PROGRAM P_ProfilePositionModeTest
VAR
	fbMoveInProfilePosition			: Motion;
	fbGetCurrentPosition			: FB_EcCoeSdoRead;
	fbGetStatusword					: FB_EcCoeSdoRead;
	fbGetPositionWindow				: FB_EcCoeSdoRead;
	fbGetPositionDemandValue		: FB_EcCoeSdoRead;
	tWaitForCurrentPosition			: TON;
	tWaitForPositionDemandValue		: TON;
	tGetStatusword					: TON;
	bGetCurrentPosition				: BOOL;
	bMove							: BOOL; 
	bExecuteTimer					: BOOL;
	bGetStatusword					: BOOL;
	bGetParameters					: BOOL;
	bSetPositioningOptionCode		: BOOL;
	bGetPositionDemandValue			: BOOL;
	bBasicOperationAbsStarted		: BOOL;
	bBasicOperationAbsFinished		: BOOL := FALSE;
	bPositioningOptionCodeSet		: BOOL;
	bTargetReached					: BOOL;
	bTestAbsolutePositioning		: BOOL;
	nTargetPosition					: DINT;
	nCurrentPosition				: DINT;
	nTargetPositionBuf				: DINT;
	nPositionDemandValue			: DINT;
	nStatusword						: UINT;
	nPositionWindow					: UDINT;
	
	
	bTest							: BOOL;
	bAusprobieren					: BOOL;
END_VAR

VAR
	bBasicOperationAbs				: BOOL;
	bBasicOperationRel				: BOOL;
	bPositioningOptionCode			: BOOL;
END_VAR

//For Test Set of Setpoints
VAR
	bSetOfSetpointFinished 			: BOOL;
	nCurrentPositionBuf				: DINT;
	bSetPointSet					: BOOL;  //For both
	bSetOfSetpoints					: BOOL;
	bStartBasicOperationAbs			: BOOL;
	bTestSetOfSetpoints				: BOOL;
	bSetOfSetpointsFinished			: BOOL;
END_VAR

//Fo Test Change Immediately
VAR
	bTestChangeImmediately			: BOOL;
	bChangeImmediatelyFinished		: BOOL;
	bChangeImmediately				: BOOL;
END_VAR

//For test of relative Positioninig
VAR
	tSetPositioningOptionCode		: TON;
	fbSetPositioningOptionCode		: FB_EcCoeSdoWrite;
	bTestRelativePositioning		: BOOL;
	bRelativePositioningFinished	: BOOL;
	nPositioningOptionCode			: DINT;
	nCounter						: DINT;
END_VAR

tWaitForCurrentPosition(IN := bGetCurrentPosition,
							PT := T#10MS);
tGetStatusword(IN := bGetStatusword,
					PT := T#500MS);	
tSetPositioningOptionCode(IN := bSetPositioningOptionCode,
							PT := T#125MS);		
tWaitForPositionDemandValue(IN := bGetPositionDemandValue,
							PT := T#125MS);
IF tWaitForCurrentPosition.Q THEN
	bGetCurrentPosition := FALSE;
ELSE
	bGetCurrentPosition := TRUE;		
END_IF
fbMoveInProfilePosition(sNetID := GVL.sNetId,
						nSlaveAddr := GVL.nSlaveAddr,
						nTargetPosition := nTargetPosition,
						bMove := bMove);
fbGetStatusword(sNetId := GVL.sNetId,
				nSlaveAddr := GVL.nSlaveAddr,
				nIndex := 16#6041,
				nSubindex := 0,
				pDstBuf := ADR(nStatusWord),
				cbBufLen := SIZEOF(nStatusWord),
				bExecute := bGetStatusword);
fbGetCurrentPosition(sNetId := GVL.sNetId,
						nSlaveAddr := GVL.nSlaveAddr,
						nIndex := 16#6064,
						nSubIndex := 0,
						pDstBuf := ADR(nCurrentPosition),
						cbBufLen := SIZEOF(nCurrentPosition),
						bExecute := bGetCurrentPosition);
fbGetPositionWindow(sNetId := GVL.sNetId,
					nSlaveAddr := GVL.nSlaveAddr,
					nIndex := 16#6067,
					nSubIndex := 0,
					pDstBuf := ADR(nPositionWindow),
					cbBufLen := SIZEOF(nPositionWindow),
					bExecute := bGetParameters);
fbGetPositionDemandValue(sNetId := GVL.sNetId,
							nSlaveAddr := GVL.nSlaveAddr,
							nIndex := 16#60FC,
							nSubIndex := 0,
							pDstBuf := ADR(nPositionDemandValue),
							cbBufLen := SIZEOF(nPositionDemandValue),
							bExecute := bGetPositionDemandValue);
fbSetPositioningOptionCode(sNetId := GVL.sNetId,
							nSlaveAddr := GVL.nSlaveAddr,
							nIndex := 16#60F2,
							nSubindex := 0,
							pSrcBuf := ADR(nPositioningOptionCode),
							cbBufLen := SIZEOF(nPositioningOptionCode),
							bExecute := bSetPositioningOptionCode);
bGetParameters := TRUE;

IF bStartBasicOperationAbs THEN					
	//Basic Operation
	//Set-point is applied to the device
	//Move to absolute position is tested
	//Wait until Target reach Bit is set
	//Control if position is within error window
	
	//Target shall be an absolute value
	MAIN.Controlword.6 := 0;

	//Operation has not yet started and we are sure that initial position is obtained
	IF NOT bBasicOperationAbsStarted THEN
		nTargetPosition := nCurrentPosition + 5000000;
		//Start absolute positioning
		bMove := TRUE;	
		bBasicOperationAbsStarted := TRUE;
	END_IF
					
	//Target reached?
	bGetStatusword := TRUE;
	IF tGetStatusword.Q THEN
		IF NOT nStatusword.10 THEN
			bGetStatusword := FALSE;
		ELSIF ((nCurrentPosition >= nTargetPosition - nPositionWindow)
				AND (nCurrentPosition <= nTargetPosition + nPositionWindow)) 
				AND fbMoveInProfilePosition.bStartPositioning THEN
			//absolute Positionining
			bBasicOperationAbs := TRUE;
			bBasicOperationAbsFinished := TRUE;
			bStartBasicOperationAbs := FALSE;
		ELSIF fbMoveInProfilePosition.bStartPositioning THEN
			bBasicOperationAbs := FALSE;
			bBasicOperationAbsFinished := TRUE;
			bStartBasicOperationAbs := FALSE;
		END_IF
		bGetStatusword := FALSE;
	END_IF
END_IF

//Test SetOfSetpoints
IF bTestSetOfSetpoints AND bBasicOperationAbsFinished AND NOT bSetOfSetpointsFinished THEN
	IF NOT bSetPointSet THEN
		MAIN.Controlword.5 := 0;
		nTargetPosition := nCurrentPosition + 100000000;
		nTargetPositionBuf := nTargetPosition;
		nCurrentPositionBuf := nCurrentPosition + 10000000/2;
		bSetPointSet := TRUE;
	END_IF
	IF (nCurrentPosition > nCurrentPositionBuf) AND bSetPointSet THEN
		nTargetPosition := nCurrentPositionBuf - 10000000/2;
	END_IF
	bSetOfSetpoints := TestChangeOfSetpoints(bActive => bSetOfSetpointsFinished);
	IF bSetOfSetpointsFinished THEN
		bSetPointSet := FALSE;
	END_IF
END_IF

//Change Immediately
IF bTestChangeImmediately AND bSetOfSetpointsFinished AND NOT bChangeImmediatelyFinished THEN
	IF NOT bSetPointSet THEN
		MAIN.Controlword.5 := 1;
		nTargetPosition := nCurrentPosition + 100000000;
		nTargetPositionBuf := nTargetPosition;
		nCurrentPositionBuf := nCurrentPosition + 10000000/2;
		bSetPointSet := TRUE;
	END_IF
	IF (nCurrentPosition > nCurrentPositionBuf) AND bSetPointSet THEN
		nTargetPosition := nCurrentPositionBuf - 10000000/2;
	END_IF
	bChangeImmediately := NOT TestChangeOfSetpoints(bActive => bChangeImmediatelyFinished);
END_IF

//Test relative positioning:
//Bit 6 of Controlword is set to 1

IF bTestRelativePositioning THEN
	MAIN.Controlword.6 := 1;
	//positioning option code: 0
	//Positioning moves shall be performed relative to the preciding
	//target position
	IF nCounter = 0 THEN
		nPositioningOptionCode := 0;
		IF tSetPositioningOptionCode.Q THEN
			nTargetPosition := 5000000;
		END_IF
		
		nCounter := nCounter + 1;
	END_IF

	//positioning option code: 2#0001
	//Positioning moves shall be performed relative to the actual
	//positioning demand value (16#60FC)
	
	//positioning option code : 2#0010
	//Positioning moves shall be performed relative to the position
	//actual value (16#6064)
END_IF

METHOD TestChangeOfSetpoints : BOOL
VAR_OUTPUT
	bActive		: BOOL;
END_VAR
IF ((nCurrentPosition >= nTargetPositionBuf - nPositionWindow)
	AND (nCurrentPosition <= nTargetPositionBuf + nPositionWindow)) THEN
	bActive := TRUE;
	bSetOfSetPointsFinished := TRUE;
ELSIF ((nCurrentPosition >= nTargetPosition - nPositionWindow)
	AND (nCurrentPosition <= nTargetPosition + nPositionWindow)) THEN
	TestChangeOfSetpoints := FALSE;
	bActive := TRUE;
END_IF
END_METHOD

END_PROGRAM

(* stored: Version 1.1.0.1, ProductVersion 3.1.4024.11
   POU P_ProfilePositionModeTest: Id {899bc5f3-4f5f-4eaa-beb6-c92d972467a4}, SpecialFunc None
   Method TestChangeOfSetpoints: Id {15b5872a-9abe-416f-a38b-72ef3f958d08} *)
